// TIA Portal V17 export
// export: Created 2022-05-07T16:38:46.0858554Z, ExportSetting WithDefaults, DisplayName Totally Integrated Automation Portal, DisplayVersion V17 Update 3, DisplayName TIA Portal Openness, DisplayVersion V17 Update 3, DisplayName TIA Portal Version Control Interface, DisplayVersion V17, DisplayName TIA Portal Test Suite Advanced, DisplayVersion V17 Update 1, DisplayName SINAMICS Startdrive Advanced, DisplayVersion V17 Update2, DisplayName SINAMICS Startdrive G130, G150, S120, S150, SINAMICS MV, S210, DisplayVersion V17 Update2, DisplayName SINAMICS Startdrive G110M, G120, G120C, G120D, G120P, G115D, DisplayVersion V17 Update2, DisplayName STEP 7 Professional, DisplayVersion V17 Update 3, DisplayName STEP 7 Safety, DisplayVersion V17, DisplayName WinCC UA Professional, DisplayVersion V17 Update 3
ORGANIZATION_BLOCK "Main"   // OB1, LAD, ProgramCycle
TITLE = "Main Program Sweep (Cycle)"
{ S7_Optimized_Access := 'TRUE' }
VERSION : 0.1
// stored: AutoNumber true, IsIECCheckEnabled false, SetENOAutomatically false
   VAR_INPUT
      Initial_Call : Bool;   // Initial call of this OB
      Remanence : Bool;   // =True, if remanent data are available
   END_VAR
BEGIN

REGION Network 1 (SCL): FORZAMENTI

   //"E0.0 FC HOMING MS" := TRUE;
END_REGION

REGION Network 2 (SCL): LANCIO BLOCCHI

   "RESET_GENERALE"("FirstScan");
   "RESET_ALLA"("RESET_ALLARMI");


   "FB_STATI_MACCHINA_DB"();

   // CICLI
   "FB_RIPRISTINO_GEN_DB"();

   "FB_RIPRISTINO_MR_DB"();
   "FB_RIPRISTINO_MA_DB"();
   "FB_RIPRISTINO_MS_DB"();
   "FB_RIPRISTINO_ME_DB"();

   "FB_CICLO_DB"();

   "FB_ORG_ASSI_DB"();

   "ALLARMI_DB"();
END_REGION
END_ORGANIZATION_BLOCK
